SUBAPPLICATION Uebung_204c_AX (* Interlock: ILOCK_CONFLICT_TRIP_PROTECT_AX (Trip bei Konflikt UND Schutzzeit nach Freigabe, via Adapter) *)
  (* Standard: 61499-2; Description: Copyright (c) 2026 Meisterschulen am Ostbahnhof This program and the accompanying materials are made available under the terms of the Eclipse Public License 2.0 which is available at https://www.eclipse.org/legal/epl-2.0/ SPDX-License-Identifier: EPL-2.0 *)
  (* Version 1.0, 2026-09-07, Franz Höpfinger, Meisterschulen am Ostbahnhof, initial API and implementation and/or initial documentation *)
  PACKAGE Uebungen;
  IMPORT logiBUS::io::DI::logiBUS_DI::Input_I1;
  IMPORT logiBUS::io::DI::logiBUS_DI::Input_I2;
  IMPORT logiBUS::io::DI::logiBUS_DI::Input_I3;
  IMPORT logiBUS::io::DI::logiBUS_DI_Events::BUTTON_SINGLE_CLICK;
  IMPORT logiBUS::io::DQ::logiBUS_DO::Output_Q1;
  IMPORT logiBUS::io::DQ::logiBUS_DO::Output_Q2;
  IMPORT logiBUS::io::DQ::logiBUS_DO::Output_Q4;
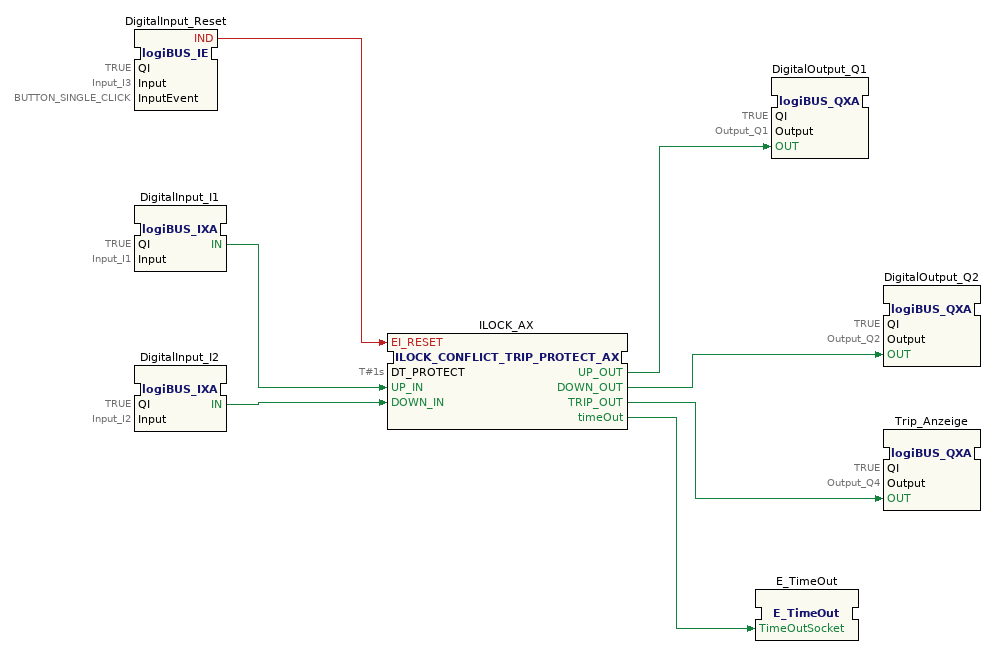
  (* Gegenueber Uebung_204_AX (ILOCK_CONFLICT_TRIP_AX): nach Freigabe des aktiven Eingangs wird DT_PROTECT (hier 1s) abgewartet, bevor eine neue Richtung (oder erneut TRIP, falls waehrenddessen der andere Eingang aktiviert wurde) uebernommen wird - dieselbe Schutzzeit-Logik wie bei ILOCK_SWITCH_PROTECT_AX (Uebung_205_AX), hier kombiniert mit der TRIP-Semantik. *)
  FBS
    DigitalInput_I1 : logiBUS::io::DI::logiBUS_IXA(QI := TRUE, Input := Input_I1);
    DigitalInput_I2 : logiBUS::io::DI::logiBUS_IXA(QI := TRUE, Input := Input_I2);
    DigitalInput_Reset : logiBUS::io::DI::logiBUS_IE(QI := TRUE, Input := Input_I3, InputEvent := BUTTON_SINGLE_CLICK);
    ILOCK_AX : logiBUS::signalprocessing::interlock::ILOCK_CONFLICT_TRIP_PROTECT_AX(DT_PROTECT := T#1s);
    DigitalOutput_Q1 : logiBUS::io::DQ::logiBUS_QXA(QI := TRUE, Output := Output_Q1);
    DigitalOutput_Q2 : logiBUS::io::DQ::logiBUS_QXA(QI := TRUE, Output := Output_Q2);
    Trip_Anzeige : logiBUS::io::DQ::logiBUS_QXA(QI := TRUE, Output := Output_Q4);
    E_TimeOut : iec61499::events::E_TimeOut;
  END_FBS
  EVENT_CONNECTIONS
    DigitalInput_Reset.IND TO ILOCK_AX.EI_RESET;
  END_CONNECTIONS
  ADAPTER_CONNECTIONS
    DigitalInput_I1.IN TO ILOCK_AX.UP_IN;
    DigitalInput_I2.IN TO ILOCK_AX.DOWN_IN;
    ILOCK_AX.UP_OUT TO DigitalOutput_Q1.OUT;
    ILOCK_AX.DOWN_OUT TO DigitalOutput_Q2.OUT;
    ILOCK_AX.TRIP_OUT TO Trip_Anzeige.OUT;
    ILOCK_AX.timeOut TO E_TimeOut.TimeOutSocket;
  END_CONNECTIONS
END_SUBAPPLICATION
